Fanuc KAREL source: ko00086.KL

-- PROVISIONAL review KL for V770-1; original PC SHA256 4cdc32f16518e5b0e84f82798995b4d2b351b7c7b1035f8be42da88fa4ddcc43
-- Incomplete behavior may be omitted. Consult companion uncertainty JSON. Do not deploy.
PROGRAM KO00086
%NOLOCKGROUP
BEGIN
  -- UNRESOLVED_PC offsets 5-12; opcodes 9D,23
  -- UNRESOLVED_PC offsets 17-69; opcodes 27,27,49,7E,AD,27,49,7E,AD,22,31,7E,4A
  -- UNRESOLVED_PC offsets 74-78; opcodes 7F
END KO00086
